Staubli VAL3: kernel.dtx

bool bEdge[5]
bool bEmergency
bool bErrorLoading
bool bHold
bool bPowered
bool bQuit
bool bRestartMove
bool bTaskPoint
bool bTimeOut
bool bWait
num nCycleStep = 4
num nLastWorkingM = 1
num nPLCClock = 7973.286
num nRemoteClock = 7973.286
num nRemoteID = -1
num nTimeOut = 10
progItem pProg
  [0]
    InstrItem iEvent
      [0]
        string sData
        string sType
    string sID
string language
string sInstr
string sItem = "JOINT @HOME"
string sMessage
string sName
string sPageLoad
string sPath
string sPathInstr
string sPathTemplate = "Disk://kernel/template/"
string sRemoteID
string sVersion[13]
  [0] = "VAL3 - s6.3.1"
  [1] = "Option testMode - demo"
  [2] = "Option valPlast - demo"
  [3] = "Configuration - D24265574A"
  [4] = "SerialNumber - ?"
  [5] = "Arm - tx90-S1-R4"
  [6] = "ArmSerialNumber - ?"
  [7] = "EP - s6.3"
  [8] = "SCA - s6.3"
  [9] = "PLC - s6.3"
  [10] = "Options - s6.3"
  [11] = "Relbo - s6.2"
  [12] = "Relbo - s5.3.2"
